(* PLC project Tc2_Coupler.CouplerReset Demo, tc3-libraries-kb TwinCAT 3.1 *)
(* stored: creationDateTime 2026-05-10T09:00:00, modificationDateTime 2026-05-10T09:00:00 *)

PROGRAM P_Demo_CouplerReset
  VAR
    fbCouplerReset : CouplerReset;  (* Function blocks 实例 *)
    arg_STATE : PLCINTFSTRUCT;  (* VAR_INPUT STATE: 2-byte PLC interface 状态字（链接到 IO） *)
    arg_START : BOOL;  (* VAR_INPUT START: 上升沿触发复位 *)
    arg_TMOUT : TIME;  (* VAR_INPUT TMOUT: 执行超时 *)
    out_CONTROL : PLCINTFSTRUCT;  (* VAR_OUTPUT CONTROL: 2-byte PLC interface 控制字（链接到 IO） *)
    out_BUSY : BOOL;  (* VAR_OUTPUT BUSY: 执行中 *)
    out_ERR : BOOL;  (* VAR_OUTPUT ERR: 执行出错 *)
    out_ERRID : UDINT;  (* VAR_OUTPUT ERRID: 错误号 *)
  END_VAR

            // ============================================================
// Tc2_Coupler.CouplerReset 演示程序
// ============================================================
// 场景：K-bus 异常时通过 PLC 远程复位耦合器
// 验证步骤：
//   1. 引用 Tc2_Coupler（及其依赖：Tc2_System 等）
//   2. 编译 + 登录
//   3. 在线监视各 out_* 输出
//   4. 必要时按场景给 arg_* 输入赋值（详见 doc.md 的'使用注意'）
// ============================================================

fbCouplerReset(
    STATE := arg_STATE,
    START := arg_START,
    TMOUT := arg_TMOUT,
    CONTROL => out_CONTROL,
    BUSY => out_BUSY,
    ERR => out_ERR,
    ERRID => out_ERRID
);

          
END_PROGRAM
